{attribute addProperty BoxType "EL7031-0000-0016"}
{attribute addProperty Id "StatusAT %I*Status_B570DD451620Counter_valueAT %I*UINT16217Latch_valueAT %I*UINT16218"}
{attribute addProperty CRC "3967730042"}
{attribute addProperty SizeInBites "48"}
{attribute addProperty SizeInBytes "6"}
TYPE ENC_Status_compact_EC7EC17A :
STRUCT
	{attribute addProperty Name "Status"}
	Status AT %I* : Status_B570DD45;
	{attribute addProperty Name "Counter_value"}
	Counter_value AT %I* : UINT;
	{attribute addProperty Name "Latch_value"}
	Latch_value AT %I* : UINT;
END_STRUCT
END_TYPE

(* stored: Version 1.2.0.0, ProductVersion 3.1.4024.9
   DUT ENC_Status_compact_EC7EC17A: Id {6d938238-485a-4122-839c-33501303f63f} *)
